// TIA Portal project "Conveyor-Based Bottle Filling and Capping" (V17)
// Bottle Line Control
// Bottles move along a conveyor, then gets filled in 15 seconds and then capped for 10 seconds only when a sensor detects the bottle.
// After that the conveyors moves again.

(* hardware
DEVICE "S7-1200 station_1"  S7-1200 Station
   slot 0: "Rack_0"  S7-1200 Rack  Rack  V1.0
   slot 1: "PLC_1"  CPU 1212C AC/DC/Rly  6ES7 212-1BE40-0XB0  V4.5
*)

// ===== PLC "PLC_1"  CPU 1212C AC/DC/Rly =====

VAR_GLOBAL   // PLC tag table "Default tag table"
   "sensor" AT %I0.1 : Bool;
   "Conveyor" AT %Q0.0 : Bool;
   "Fill valve/pump" AT %Q0.1 : Bool;
   "Capper actuator" AT %Q0.2 : Bool;
   "Start_station" AT %I0.0 : Bool;
   "Tag_1" AT %M0.0 : Bool;
   "Tag_2" AT %M0.1 : Bool;
   "Tag_3" AT %M0.2 : Bool;
   "Tag_4" AT %M0.3 : Bool;
END_VAR

// folder: System blocks/Program resources

DATA_BLOCK "IEC_Timer_0_DB"   // DB1
{ S7_Optimized_Access := 'TRUE' }
AUTHOR : Simatic
FAMILY : IEC
NAME : IEC_TMR
VERSION : 1.0
// stored: InstanceOfName IEC_TIMER
"IEC_TIMER"
BEGIN
END_DATA_BLOCK

DATA_BLOCK "IEC_Timer_0_DB_1"   // DB2
{ S7_Optimized_Access := 'TRUE' }
AUTHOR : Simatic
FAMILY : IEC
NAME : IEC_TMR
VERSION : 1.0
// stored: InstanceOfName IEC_TIMER
"IEC_TIMER"
BEGIN
END_DATA_BLOCK

DATA_BLOCK "IEC_Timer_0_DB_2"   // DB3
{ S7_Optimized_Access := 'TRUE' }
AUTHOR : Simatic
FAMILY : IEC
NAME : IEC_TMR
VERSION : 1.0
// stored: InstanceOfName IEC_TIMER
"IEC_TIMER"
BEGIN
END_DATA_BLOCK

DATA_BLOCK "IEC_Timer_0_DB_3"   // DB4
{ S7_Optimized_Access := 'TRUE' }
AUTHOR : Simatic
FAMILY : IEC
NAME : IEC_TMR
VERSION : 1.0
// stored: InstanceOfName IEC_TIMER
"IEC_TIMER"
BEGIN
END_DATA_BLOCK

// folder: (top level)

ORGANIZATION_BLOCK "Main"   // OB1, LAD, ProgramCycle
TITLE = "Main Program Sweep (Cycle)"
{ S7_Optimized_Access := 'TRUE' }
VERSION : 0.1
   VAR_INPUT
      Initial_Call : Bool;   // Initial call of this OB
      Remanence : Bool;   // =True, if remanent data are available
   END_VAR
   VAR_TEMP   // added for the SCL form of the ladder/FBD networks
      _w1 : Bool;
      _w2 : Bool;
   END_VAR
BEGIN

REGION Network 1
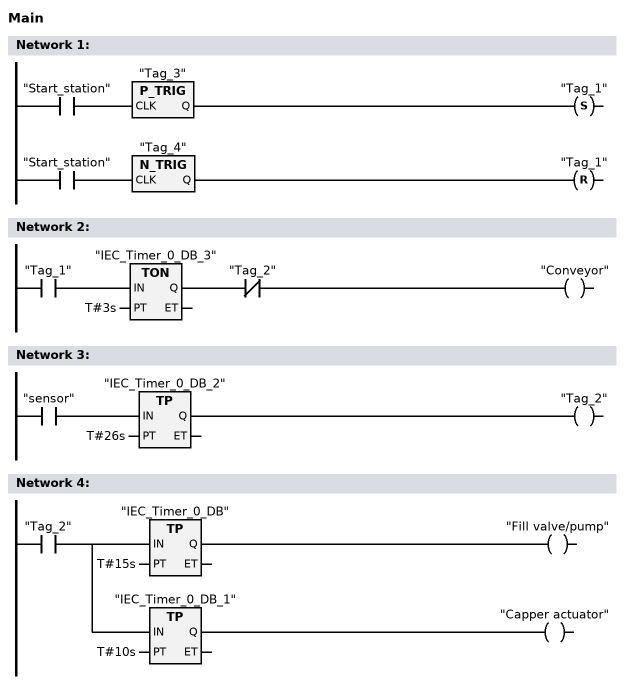
   RUNG wire#powerrail
      Contact( "Start_station" )
      P_Trig( "Tag_3" )
      S_Coil( "Tag_1" )
   END_RUNG
   RUNG wire#powerrail
      Contact( "Start_station" )
      N_Trig( "Tag_4" )
      R_Coil( "Tag_1" )
   END_RUNG
   // the same network as SCL:
   #_w1 := "Start_station" AND NOT "Tag_3";   // rising edge
   "Tag_3" := "Start_station";
   IF #_w1 THEN "Tag_1" := TRUE; END_IF;
   #_w2 := NOT "Start_station" AND "Tag_4";   // falling edge
   "Tag_4" := "Start_station";
   IF #_w2 THEN "Tag_1" := FALSE; END_IF;
END_REGION

REGION Network 2
   "IEC_Timer_0_DB_3".TON(IN := "Tag_1", PT := T#3s);
   "Conveyor" := "IEC_Timer_0_DB_3".Q AND NOT "Tag_2";
END_REGION

REGION Network 3
   "IEC_Timer_0_DB_2".TP(IN := "sensor", PT := T#26s);
   "Tag_2" := "IEC_Timer_0_DB_2".Q;
END_REGION

REGION Network 4
   "IEC_Timer_0_DB".TP(IN := "Tag_2", PT := T#15s);
   "Fill valve/pump" := "IEC_Timer_0_DB".Q;
   "IEC_Timer_0_DB_1".TP(IN := "Tag_2", PT := T#10s);
   "Capper actuator" := "IEC_Timer_0_DB_1".Q;
END_REGION
END_ORGANIZATION_BLOCK